FUNCTION Safety : BOOL
VAR_INPUT
	Obstacle : BOOL;
END_VAR
VAR
END_VAR

IF Obstacle =TRUE THEN		// IF there is an obstacle it is not safe
	Safety := FALSE;
	ELSE
		Safety :=TRUE;		// If there is not an obstacle it is safe
END_IF

END_FUNCTION

(* stored: Version 1.1.0.1, ProductVersion 3.1.4024.15
   POU Safety: Id {c033ce95-c04b-4aed-9409-cf1159682b9d}, SpecialFunc None *)
